// TIA Portal V16 export
// export: Created 2021-06-17T11:14:32.0828374Z, ExportSetting WithDefaults, DisplayName Totally Integrated Automation Portal, DisplayVersion V16 Update 4, DisplayName TIA Portal Version Control Interface, DisplayVersion V16 Update 2, DisplayName TIA Portal Openness, DisplayVersion V16 Update 4, DisplayName SINAMICS Startdrive Advanced, DisplayVersion V16 Update 5, DisplayName SINAMICS Startdrive G130, G150, S120, S150, SINAMICS MV, S210, DisplayVersion V16 Update 5, DisplayName SINAMICS Startdrive G110M, G120, G120C, G120D, G120P, G115D, DisplayVersion V16 Update 5, DisplayName STEP 7 Professional, DisplayVersion V16 Update 4, DisplayName SIMATIC Energy Suite, DisplayVersion V16 Update 4, DisplayName STEP 7 Safety, DisplayVersion V16, DisplayName WinCC Advanced / Unified PC, DisplayVersion V16 Update 4, DisplayName SIMATIC Visualization Architect, DisplayVersion V16 Update 1
DATA_BLOCK "Runtime_test_1_DB"   // DB5
VERSION : 0.1
// stored: AutoNumber true, DBAccessibleFromOPCUA true, InstanceOfName Runtime_test_1, InstanceOfType FB
"Runtime_test_1"
   // VAR
   //    FB_LTIME_opt : LReal;
   //    FB_LTIME_notopt : LReal;
   //    MEM_RUNTIME_opt : LReal;
   //    MEM_RUNTIME_notopt : LReal;
   //    FB_LTIME_notopt_tmp : LReal;
   //    FB_LTIME_opt_tmp : LReal;
   //    opimized { ExternalAccessible := 'False'; ExternalVisible := 'False'; ExternalWritable := 'False'} : Array[0..500] of "UDT_ACB_ETI";
   // END_VAR
BEGIN
END_DATA_BLOCK
